SYSTEM MPP_VIEWL (* View test configuration for Mini Pulp Process *)
  (* Standard: IEC 61499 *)
  (* Version 0.5, 2006-12-08, JHC, Holobloc Inc, Adjusted for new IN_PAINT element (textured painting). *)
  (* Version 0.4, 2006-11-17, JHC, Holobloc Inc, Added colors for valves, pumps + pipes. *)
  (* Version 0.3, 2006-11-16, JHC, Holobloc Inc, Added T300 colors. *)
  (* Version 0.2, 2006-11-07, JHC, Holobloc Inc, Added Tanks + HMI elements. *)
  (* Version 0.1, 2006-08-19, JHC, Holobloc Inc, Added E100 (Heater). *)
  (* Version 0.0, 2006-08-19, JHC, Holobloc Inc, Adapted for inclusion of Nodes in GRAPH_RESOURCE.GRAPH file. *)
  DEVICE HMI : FRAME_DEVICE(BOUNDS := [0,50,390,650])
    RESOURCE ACTUATORS : PANEL_RESOURCE(COLS := 3) (* Valves and Pumps *)
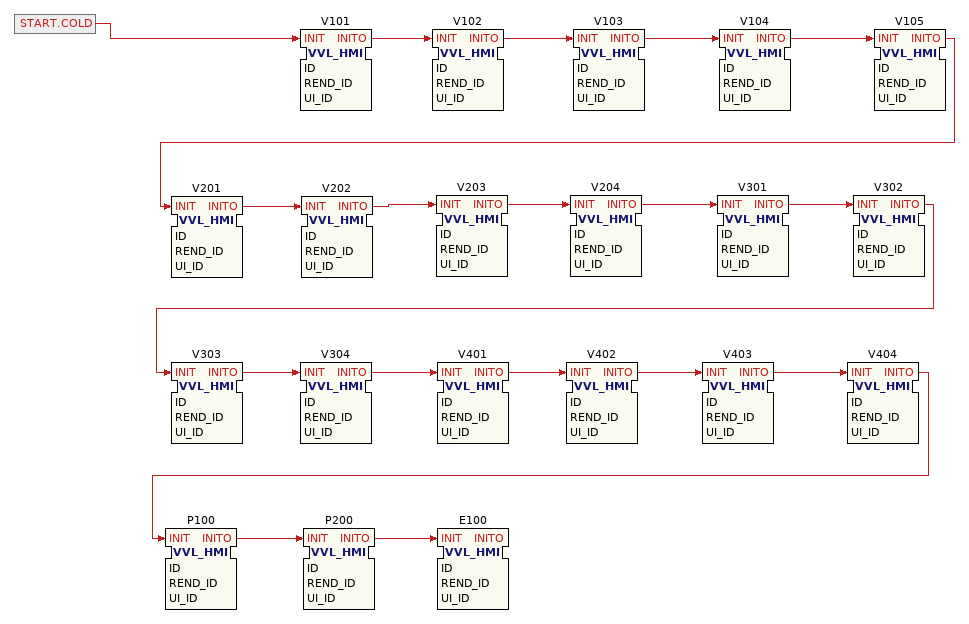
      FBS
        V101 : VVL_HMI;
        V204 : VVL_HMI;
        V103 : VVL_HMI;
        V102 : VVL_HMI;
        V104 : VVL_HMI;
        V105 : VVL_HMI;
        V201 : VVL_HMI;
        V202 : VVL_HMI;
        V203 : VVL_HMI;
        V301 : VVL_HMI;
        V302 : VVL_HMI;
        V303 : VVL_HMI;
        V304 : VVL_HMI;
        V401 : VVL_HMI;
        V402 : VVL_HMI;
        V403 : VVL_HMI;
        V404 : VVL_HMI;
        P100 : VVL_HMI;
        P200 : VVL_HMI;
        E100 : VVL_HMI;
      END_FBS
      EVENT_CONNECTIONS
        START.COLD TO V101.INIT;
        V101.INITO TO V102.INIT;
        V102.INITO TO V103.INIT;
        V103.INITO TO V104.INIT;
        V104.INITO TO V105.INIT;
        V105.INITO TO V201.INIT;
        V201.INITO TO V202.INIT;
        V202.INITO TO V203.INIT;
        V203.INITO TO V204.INIT;
        V204.INITO TO V301.INIT;
        V301.INITO TO V302.INIT;
        V302.INITO TO V303.INIT;
        V303.INITO TO V304.INIT;
        V304.INITO TO V401.INIT;
        V401.INITO TO V402.INIT;
        V402.INITO TO V403.INIT;
        V403.INITO TO V404.INIT;
        V404.INITO TO P100.INIT;
        P100.INITO TO P200.INIT;
        P200.INITO TO E100.INIT;
      END_CONNECTIONS
    END_RESOURCE
    RESOURCE SENSORS : PANEL_RESOURCE(COLS := 1)
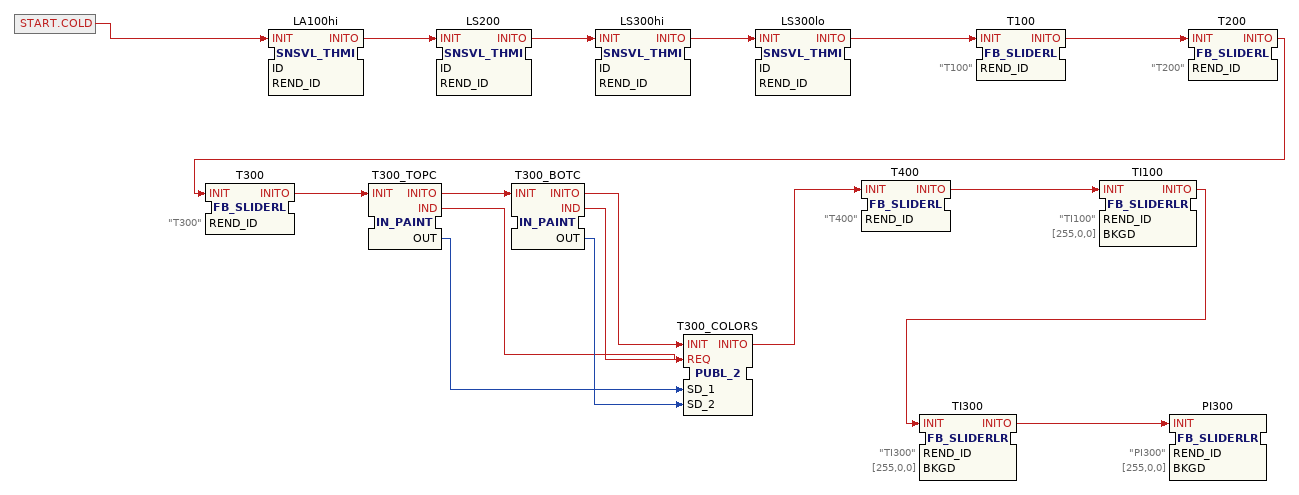
      FBS
        LA100hi : SNSVL_THMI; (* 0 = Tank 100 Overflow *)
        LS200 : SNSVL_THMI;
        LS300lo : SNSVL_THMI;
        LS300hi : SNSVL_THMI;
        T100 : FB_SLIDERL(REND_ID := "T100");
        T200 : FB_SLIDERL(REND_ID := "T200");
        T300 : FB_SLIDERL(REND_ID := "T300");
        T400 : FB_SLIDERL(REND_ID := "T400");
        PI300 : FB_SLIDERLR(REND_ID := "PI300", BKGD := [255,0,0]);
        TI300 : FB_SLIDERLR(REND_ID := "TI300", BKGD := [255,0,0]);
        TI100 : FB_SLIDERLR(REND_ID := "TI100", BKGD := [255,0,0]);
        T300_TOPC : IN_PAINT; (* T300 top (deselected) color *)
        T300_BOTC : IN_PAINT; (* T300 bottom (selected) color *)
        T300_COLORS : PUBL_2; (* T300 top, bottom colors *)
      END_FBS
      EVENT_CONNECTIONS
        START.COLD TO LA100hi.INIT;
        LA100hi.INITO TO LS200.INIT;
        T200.INITO TO T300.INIT;
        LS200.INITO TO LS300hi.INIT;
        LS300hi.INITO TO LS300lo.INIT;
        LS300lo.INITO TO T100.INIT;
        T300_TOPC.INITO TO T300_BOTC.INIT;
        T300_BOTC.INITO TO T300_COLORS.INIT;
        T300_BOTC.IND TO T300_COLORS.REQ;
        T300_COLORS.INITO TO T400.INIT;
        T300_TOPC.IND TO T300_COLORS.REQ;
        T300.INITO TO T300_TOPC.INIT;
        T100.INITO TO T200.INIT;
        T400.INITO TO TI100.INIT;
        TI100.INITO TO TI300.INIT;
        TI300.INITO TO PI300.INIT;
      END_CONNECTIONS
      DATA_CONNECTIONS
        T300_TOPC.OUT TO T300_COLORS.SD_1;
        T300_BOTC.OUT TO T300_COLORS.SD_2;
      END_CONNECTIONS
    END_RESOURCE
  END_DEVICE
  DEVICE VIEW : FRAME_DEVICE(BOUNDS := [325,50,705,650])
    RESOURCE MODE_CTL : PANEL_RESOURCE
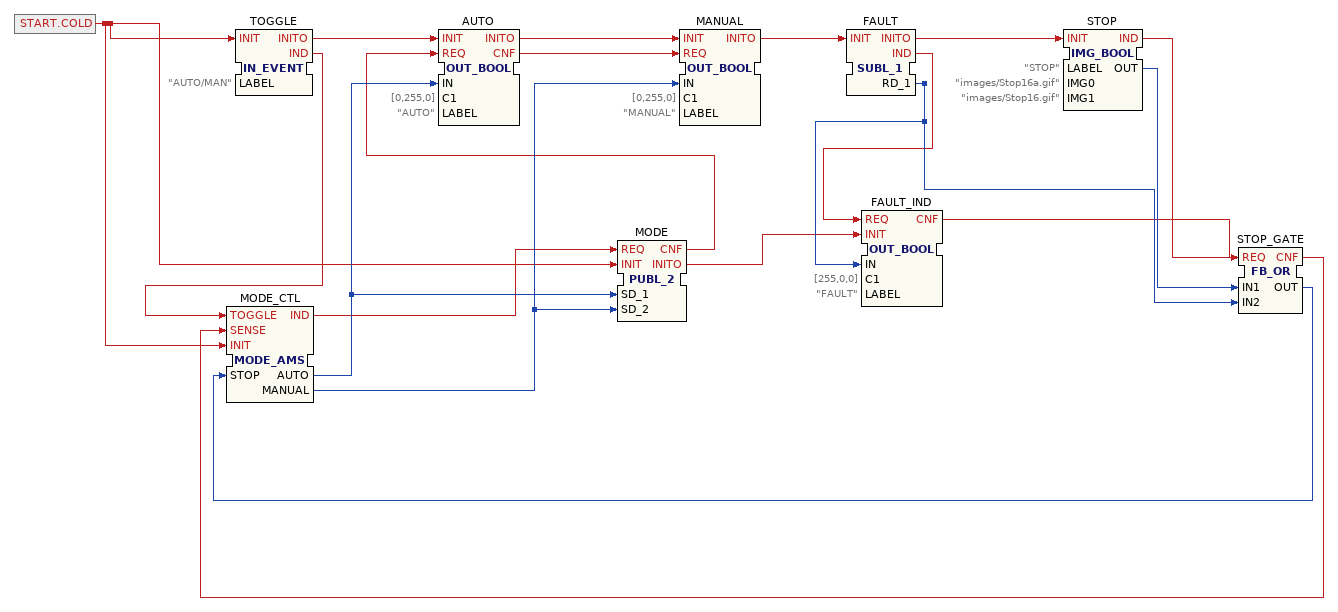
      FBS
        FAULT_IND : OUT_BOOL(C1 := [255,0,0], LABEL := "FAULT");
        FAULT : SUBL_1;
        MODE : PUBL_2;
        MODE_CTL : MODE_AMS;
        TOGGLE : IN_EVENT(LABEL := "AUTO/MAN");
        AUTO : OUT_BOOL(C1 := [0,255,0], LABEL := "AUTO");
        MANUAL : OUT_BOOL(C1 := [0,255,0], LABEL := "MANUAL");
        STOP : IMG_BOOL(LABEL := "STOP", IMG0 := "images/Stop16a.gif", IMG1 := "images/Stop16.gif");
        STOP_GATE : FB_OR;
      END_FBS
      EVENT_CONNECTIONS
        START.COLD TO TOGGLE.INIT;
        TOGGLE.INITO TO AUTO.INIT;
        AUTO.INITO TO MANUAL.INIT;
        AUTO.CNF TO MANUAL.REQ;
        MODE_CTL.IND TO MODE.REQ;
        TOGGLE.IND TO MODE_CTL.TOGGLE;
        MODE.CNF TO AUTO.REQ;
        STOP.IND TO STOP_GATE.REQ;
        MANUAL.INITO TO FAULT.INIT;
        FAULT.INITO TO STOP.INIT;
        FAULT.IND TO FAULT_IND.REQ;
        FAULT_IND.CNF TO STOP_GATE.REQ;
        STOP_GATE.CNF TO MODE_CTL.SENSE;
        START.COLD TO MODE.INIT;
        MODE.INITO TO FAULT_IND.INIT;
        START.COLD TO MODE_CTL.INIT;
      END_CONNECTIONS
      DATA_CONNECTIONS
        FAULT.RD_1 TO FAULT_IND.IN;
        MODE_CTL.AUTO TO MODE.SD_1;
        MODE_CTL.MANUAL TO MODE.SD_2;
        MODE_CTL.AUTO TO AUTO.IN;
        MODE_CTL.MANUAL TO MANUAL.IN;
        STOP.OUT TO STOP_GATE.IN1;
        FAULT.RD_1 TO STOP_GATE.IN2;
        STOP_GATE.OUT TO MODE_CTL.STOP;
      END_CONNECTIONS
    END_RESOURCE
    RESOURCE GRAPH : GRAPH_RESOURCE(GRAPH := "batch/MPP_GRAPH.xml")
    END_RESOURCE
  END_DEVICE
END_SYSTEM
